{attribute 'GeneratedUsingTerminal: EJ9576-0000-0018'}
{attribute addProperty BoxType "EJ9576-0000-0018"}
{attribute addProperty Id "BCT_InputsAT %I*BCT_Inputs_8E55234D16WcStateAT %I*WcState_9091E0EB2InfoDataAT %I*InfoData_32EB74EA10"}
{attribute addProperty CRC "1836276170"}
{attribute addProperty Size "28"}
TYPE EJ9576_6D7359CA EXTENDS EtcSlaveTerminalBase_947E5A46 :
STRUCT
	{attribute addProperty Name "BCT_Inputs"}
	BCT_Inputs : BCT_Inputs_8E55234D;
	{attribute addProperty Name "WcState"}
	WcState : WcState_9091E0EB;
	{attribute addProperty Name "InfoData"}
	InfoData : InfoData_32EB74EA;
END_STRUCT
END_TYPE

(* stored: Version 1.2.0.0, ProductVersion 3.1.4024.9
   DUT EJ9576_6D7359CA: Id {bc43dd79-cae2-4189-9de5-4763fdc5397c} *)
